{attribute 'qualified_only'}
{attribute 'strict'}
{attribute 'to_string'}
TYPE E_AXIS_SELECTOR :
(
	SELECT_INDEX,
  SELECT_AXIS_ID
);
END_TYPE

(* stored: Version 1.1.0.1, ProductVersion 3.1.4026.18
   DUT E_AXIS_SELECTOR: Id {488fac83-78dd-4907-b8e7-a4a8007f9fea} *)
